GLOBALCONSTANTS STATES (* States (Closed, Opened, Transitions) *)
  (* Standard: 61499-1; Description: Copyright (c) 2025 HR Agrartechnik GmbH This program and the accompanying materials are made available under the terms of the Eclipse Public License 2.0 which is available at https://www.eclipse.org/legal/epl-2.0/ SPDX-License-Identifier: EPL-2.0 *)
  (* Version 1.0, 2025-05-23, Franz Höpfinger, HR Agrartechnik GmbH *)
  PACKAGE logiBUS::utils::sequence::schieber::const;
  IMPORT eclipse4diac::core::TypeHash;
  VAR_GLOBAL CONSTANT
    Unknown : STRING := STRING#'Unknown';
    Closed : STRING := STRING#'Closed';
    Opening : STRING := STRING#'Opening';
    Opened : STRING := STRING#'Opened';
    Closing : STRING := STRING#'Closing';
  END_VAR
END_GLOBALCONSTANTS
